(* CoDeSys 2.3.9.25 project: fuel_oil_v1.4.4.pro *)
(* Libraries: Util.lib 18.5.10 16:14:28, STANDARD.LIB 4.10.05 12:14:46, IECSFC.LIB 13.4.06 16:51:28, ANALYZATION.LIB 5.10.99 10:05:06 *)

(* PLC configuration (modules and I/O channels)
Fast discrete inputs [I_SIMPLE_INPUT] node 0, in %IB0 out %QB0 {Filtrationtime = 10; Visibility = No}
  AT %IX0.0 [BitInput] Discrete input 1
  AT %IX0.1 [BitInput] Discrete input 2
Discrete inputs - 16 [ID130] node 1, in %IB1 out %QB1 {Filtrationtime_GeneralINP = 1; Visibility = No; PinCount = 16}
  AT %IB1.0 [ByteInput] 8 discrete inputs
  AT %IB1.1 [ByteInput] 8 discrete inputs
Fast discrete outputs [OWEN_ID570] node 2, in %IB2 out %QB2 {SafeValueBool = FALSE; SafeValueBool = FALSE; SafeValueBool = FALSE; SafeValueBool = FALSE; Visibility = No}
  AT %QX2.0 [BitOutput] go_emul
  AT %QX2.1 [BitOutput] go_mixing
  AT %QX2.2 [BitOutput] go_diesel_bio
  AT %QX2.3 [BitOutput] go_water
AT %QB3.0 [ByteOutput] 8 discrete outputs
AT %QB3.1 [ByteOutput] 2 discrete outputs
Special input [ID103] node 4, in %IB4 out %QB4 {Filtrationtime = 1000; PinCount = 1; WatchDogPeriod = 400; PollPeriod = 3000; Visibility = No}
  AT %IX4.0 [BitInput] Special input
Special output [ID104] node 5, in %IB5 out %QB5 {Visibility = No; PinCount = 1}
  AT %QX5.0 [BitOutput] Special output
ModBus (Master) [MODBUS_MASTER_ID450] node 6, in %IB6 out %QB6 {Visibility = No}
  AT %QD6.0 [DWordOutput] Last address
  AT %QW6.1 [WordOutput] Last error
  RS-485-1 [COM1_USART] node 0, in %IB6.0 out %QB6.0 {CommunicationSpeed = 11520; Parity = NO PARITY CHECK; BitLength = 8 bits; StopLength = One stop bit; InterfaceType = RS485; FrameOriented = RTU; Timeout = 0; Visibility = No}
AT %QB6.1.0 [ComChannel] Command (0xff - Start)
AT %IW6.1.0.0 [WordInput]
AT %ID6.1.1.0 [FloatInput]
TCP [TCP_ID221] node 0, in %IB7.0.0 out %QB7.0.0 {RemotePort = 502; Visibility = No}
AT %QB7.1.0 [ByteOutput]
AT %QB7.2.0 [ByteOutput]
AT %QW7.3.0 [WordOutput] flow_out
AT %QW7.4.0 [WordOutput] weight_of_emul_LAN
AT %QW7.5.0 [WordOutput] weight_of_diesel_LAN
AT %QW7.6.0 [WordOutput] weight_of_biodiesel_LAN
AT %QW7.7.0 [WordOutput] set_number_of_liters_LAN
AT %QW7.8.0 [WordOutput] time_of_mixing_first
AT %QW7.9.0 [WordOutput] weight_left_LAN
AT %QW7.10.0 [WordOutput] empty
AT %QW7.11.0 [WordOutput] empty
AT %QW7.12.0 [WordOutput] avto_LAN
AT %QW7.13.0 [WordOutput] number_of_liters_LAN
AT %QW7.14.0 [WordOutput] time_of_mixing_second
AT %QW7.15.0 [WordOutput] pusk_LAN
AT %QW7.16.0 [WordOutput] stop_LAN
AT %QD7.17.0 [FloatOutput] wight_in_barrel_LAN
AT %QD7.18.0 [FloatOutput] wight_in_barrel_for_proc
AT %QD7.19.0 [FloatOutput] wight_for_sub_2
*)

(* POU PLC_PRG, LD *)
PROGRAM PLC_PRG
VAR
(*блок запуска/остоновки/паузы*)
	psp: psp;
	pusk AT %IX1.0.1: BOOL; (*сигнал на запуск цикла*)
	pusk_LAN AT %QW7.15.0: BOOL; (*сигнал на запуск цикла со SCADA*)
	avto AT %IX1.0.3: BOOL; (*перевод системы в автоматический режим*)
	stop AT %IX1.0.2: BOOL; (*сигнал на остановку цикла*)
	stop_LAN AT %QW7.16.0: BOOL; (*сигнал на остановку цикла со SCADA*)
	pusk_prog: BOOL; (*цикл запущен*)
	stop_prog AT %QX7.1.0.0: BOOL; (*цикл остановлен*)
	pause: BOOL; (*цикл поставлен на паузу*)
	wight_in_barrel AT %ID6.1.1.0: REAL; (*вес в баке, приходящий с весов*)
	work_lamp AT %QX3.0.3: BOOL; (*выходная лампа сигнализации работы*)
	wight_in_barrel_for_proc AT %QD7.18.0: REAL; (*количество кг смеси для цикла*)
	flow_reley AT %IX1.1.4: BOOL; (*срабатывание реле протока*)
	TZ2_LAN AT %QX7.1.0.3: BOOL;
	TZ3_LAN AT %QX7.1.0.4: BOOL;
	TZ4_LAN AT %QX7.1.0.5: BOOL;
	TZ5_LAN AT %QX7.1.0.6: BOOL;
	TZ6_LAN AT %QX7.1.0.7: BOOL;
	TZ7_LAN AT %QX7.2.0.0: BOOL;
	work_lamp_LAN AT %QX7.2.0.1: BOOL; (*лампа работы для Scada*)
	wight_in_barrel_LAN AT %QD7.17.0: REAL; (*значение текущего ввеса в баке для Scada*)
	for_setpoints: REAL; (*значения для рассчета аозможности перелива*)

(*блок предотвращения перелива жидкости из бака*)
	sum_of_setpoints: sum_of_setpoints;
	more_then_need AT %QX7.2.0.2: BOOL; (*сигнализации о том, что может произойти перелив*)

(*Блок для отправки значений работы насосов в Scada*)
	move_block: move_block;
	go_emul_LAN AT %QX7.2.0.3: BOOL;
	go_diesel_bio_LAN AT %QX7.2.0.4: BOOL;
	go_water_LAN AT %QX7.2.0.5: BOOL;
	go_mixing_LAN AT %QX7.2.0.6: BOOL;
	go_disper_LAN AT %QX7.2.0.7: BOOL;
	avto_LAN AT %QW7.12.0: BOOL;

(*блок запуска процесса наполнения бака эмульсией*)
	emul: emul;
	go_emul AT %QX2.0: BOOL; (*сигнал на запуск насоса эмульсии*)
	end_work_emul: BOOL; (*блок работы насоса эмульсии завершен*)
	flow_out: BOOL; (*реле протока не сработало*)
	flow_out_LAN AT %QW7.3.0: BOOL;

(*блок запуска насоса дизель/биодизель*)
	dies_bio: dies_bio;
	go_diesel_bio AT %QX2.2: BOOL; (*сигнал на запуск насоса дизель/биодизель*)
	stop_diesel: BOOL; (*сигнал о том что, наполнение дизеля в бак окончено*)
	end_work_dies_bio AT %QX7.1.0.1: BOOL; (*блок работы насоса дизель/биодизель завершен*)
	weight_next_step: REAL; (*количество жидкости для продолжения цикла*)
	both_null: BOOL;

(*блок запуска насоса воды*)
	water: water;
	count AT %IX0.0: BOOL; (*импульсы, приходящие со счетчика воды*)
	number_of_liters_LAN AT %QW7.13.0: WORD; (*количество воды, посчитанное счетчиком воды*)
	go_water AT %QX2.3: BOOL; (*сигнал на запуск насоса воды*)
	end_work_water: BOOL; (*блок работы насоса воды завершен*)
	go_valve AT %QX3.0.5: BOOL;

(*блок управлени насосом смешивания*)
	mixing: mixing;
	go_mixing AT %QX2.1: BOOL; (*сигнал на запуск насоса смешивания*)
	end_work_mixing: BOOL; (*блок работы насоса смешивания завершен*)
	end_work_first AT %QX7.1.0.2: BOOL; (*блок работы насоса завершил первое перемешивание*)

(*блок управления насосом диспергации*)
	disper: disper;
	go_disper AT %QX3.0.0: BOOL; (*сигнал на запуск насоса смешивания*)
	end_work_disper: BOOL; (*блок работы насоса диспергации завершен*)

	TZ2 AT %IX1.0.6: BOOL;
	TZ3 AT %IX1.0.7: BOOL;
	TZ4 AT %IX1.1.0: BOOL;
	TZ5 AT %IX1.1.1: BOOL;
	TZ6 AT %IX1.1.2: BOOL;
	TZ7 AT %IX1.1.3: BOOL;
	avar_TZ: BOOL; (*сработала одна из тепловых защит*)
	weight_of_diesel_for_mix: BOOL;

	for_calculate: CTU;
	calc_trig: R_TRIG;
	wight_for_sub_1: REAL;
	wight_for_sub_2 AT %QD7.19.0: REAL;
END_VAR

VAR RETAIN PERSISTENT
	weight_of_emul_LAN AT %QW7.4.0: WORD; (*количество эмульгатора для наполнения в бак, задается из SCADA*)
	weight_of_diesel_LAN AT %QW7.5.0: WORD; (*количество дизеля для наполнения в бак, задается из SCADA*)
	weight_of_biodiesel_LAN AT %QW7.6.0: WORD; (*количество биодизеля для наполнения в бак, задается из SCADA*)
	set_number_of_liters_LAN AT %QW7.7.0: WORD; (*количество воды для наполнения в бак, задается из SCADA*)
	time_of_mixing_first AT %QW7.8.0: WORD; (*время первого смешивания*)
	weight_left_LAN AT %QW7.9.0: WORD; (*колличество, которое должно остаться в баке после диспергации*)
	time_of_mixing_second AT %QW7.14.0: WORD; (*время второго смешивания*)
END_VAR
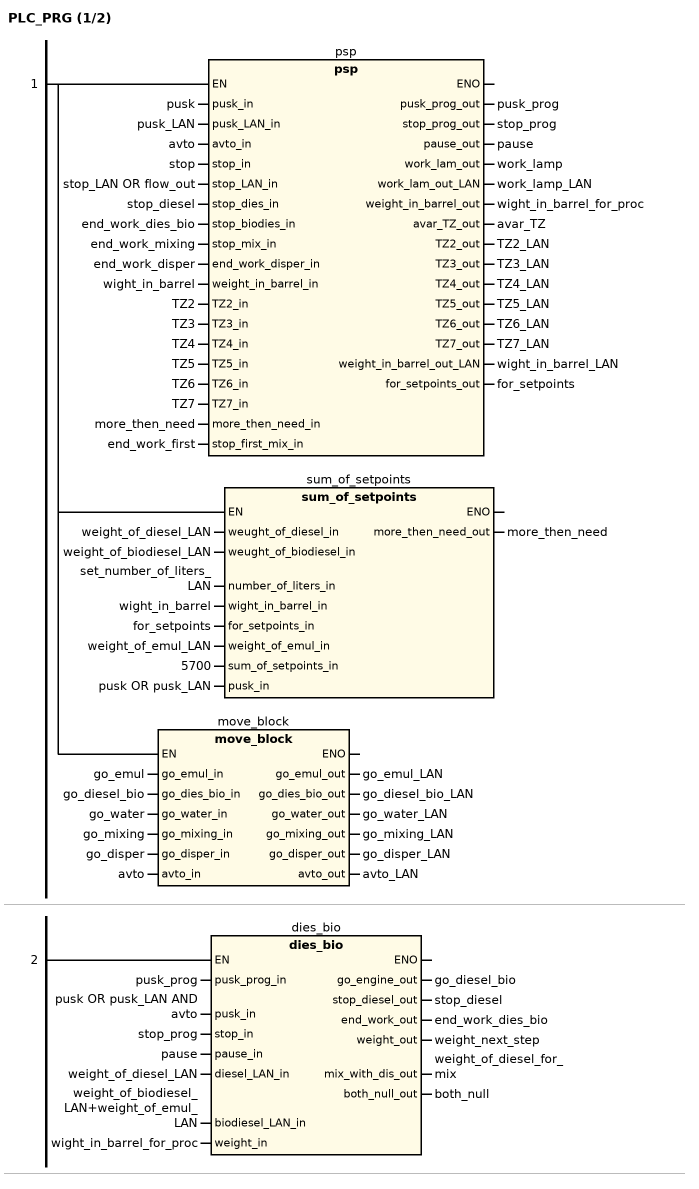
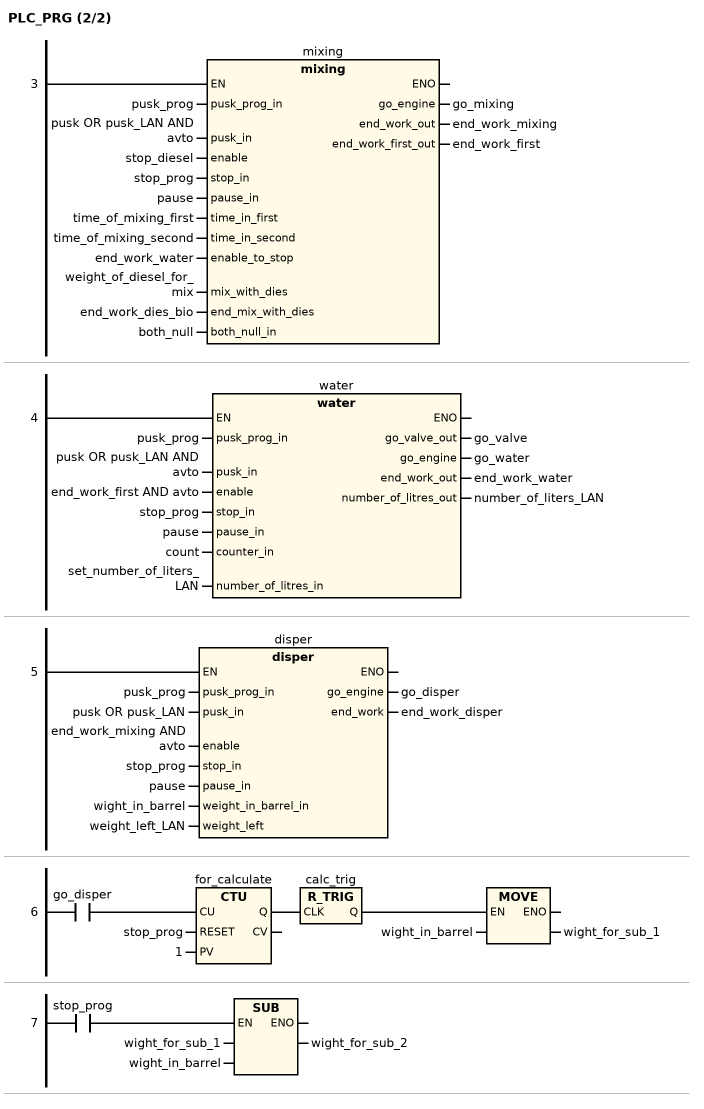
_LD_ (* Ladder Diagram *)
NETWORK 1
	*
		EN --- psp:psp(pusk_in: pusk, pusk_LAN_in: pusk_LAN, avto_in: avto, stop_in: stop, stop_LAN_in: stop_LAN OR flow_out, stop_dies_in: stop_diesel, stop_biodies_in: end_work_dies_bio, stop_mix_in: end_work_mixing, end_work_disper_in: end_work_disper, weight_in_barrel_in: wight_in_barrel, TZ2_in: TZ2, TZ3_in: TZ3, TZ4_in: TZ4, TZ5_in: TZ5, TZ6_in: TZ6, TZ7_in: TZ7, more_then_need_in: more_then_need, stop_first_mix_in: end_work_first, stop_prog_out => stop_prog, pause_out => pause, work_lam_out => work_lamp, work_lam_out_LAN => work_lamp_LAN, weight_in_barrel_out => wight_in_barrel_for_proc, avar_TZ_out => avar_TZ, TZ2_out => TZ2_LAN, TZ3_out => TZ3_LAN, TZ4_out => TZ4_LAN, TZ5_out => TZ5_LAN, TZ6_out => TZ6_LAN, TZ7_out => TZ7_LAN, weight_in_barrel_out_LAN => wight_in_barrel_LAN, for_setpoints_out => for_setpoints) => pusk_prog
		EN --- sum_of_setpoints:sum_of_setpoints(weught_of_diesel_in: weight_of_diesel_LAN, weught_of_biodiesel_in: weight_of_biodiesel_LAN, number_of_liters_in: set_number_of_liters_LAN, wight_in_barrel_in: wight_in_barrel, for_setpoints_in: for_setpoints, weight_of_emul_in: weight_of_emul_LAN, sum_of_setpoints_in: 5700, pusk_in: pusk OR pusk_LAN) => more_then_need
		EN --- move_block:move_block(go_emul_in: go_emul, go_dies_bio_in: go_diesel_bio, go_water_in: go_water, go_mixing_in: go_mixing, go_disper_in: go_disper, avto_in: avto, go_dies_bio_out => go_diesel_bio_LAN, go_water_out => go_water_LAN, go_mixing_out => go_mixing_LAN, go_disper_out => go_disper_LAN, avto_out => avto_LAN) => go_emul_LAN
NETWORK 2
	*
		EN --- dies_bio:dies_bio(pusk_prog_in: pusk_prog, pusk_in: pusk OR pusk_LAN AND avto, stop_in: stop_prog, pause_in: pause, diesel_LAN_in: weight_of_diesel_LAN, biodiesel_LAN_in: weight_of_biodiesel_LAN+weight_of_emul_LAN, weight_in: wight_in_barrel_for_proc, stop_diesel_out => stop_diesel, end_work_out => end_work_dies_bio, weight_out => weight_next_step, mix_with_dis_out => weight_of_diesel_for_mix, both_null_out => both_null) => go_diesel_bio
NETWORK 3
	*
		EN --- mixing:mixing(pusk_prog_in: pusk_prog, pusk_in: pusk OR pusk_LAN AND avto, enable: stop_diesel, stop_in: stop_prog, pause_in: pause, time_in_first: time_of_mixing_first, time_in_second: time_of_mixing_second, enable_to_stop: end_work_water, mix_with_dies: weight_of_diesel_for_mix, end_mix_with_dies: end_work_dies_bio, both_null_in: both_null, end_work_out => end_work_mixing, end_work_first_out => end_work_first) => go_mixing
NETWORK 4
	*
		EN --- water:water(pusk_prog_in: pusk_prog, pusk_in: pusk OR pusk_LAN AND avto, enable: end_work_first AND avto, stop_in: stop_prog, pause_in: pause, counter_in: count, number_of_litres_in: set_number_of_liters_LAN, go_engine => go_water, end_work_out => end_work_water, number_of_litres_out => number_of_liters_LAN) => go_valve
NETWORK 5
	*
		EN --- disper:disper(pusk_prog_in: pusk_prog, pusk_in: pusk OR pusk_LAN, enable: end_work_mixing AND avto, stop_in: stop_prog, pause_in: pause, weight_in_barrel_in: wight_in_barrel, weight_left: weight_left_LAN, end_work => end_work_disper) => go_disper
NETWORK 6
	[go_disper] - for_calculate:CTU(CU: *, RESET: stop_prog, PV: 1) - calc_trig:R_TRIG(CLK: *)
		EN --- MOVE(wight_in_barrel) => wight_for_sub_1
NETWORK 7
	[stop_prog]
		EN --- SUB(wight_for_sub_1, wight_in_barrel) => wight_for_sub_2
_END_LD_
(* the same logic as Structured Text *)
(* Network 1 *)
psp(pusk_in := pusk, pusk_LAN_in := pusk_LAN, avto_in := avto, stop_in := stop, stop_LAN_in := stop_LAN OR flow_out, stop_dies_in := stop_diesel, stop_biodies_in := end_work_dies_bio, stop_mix_in := end_work_mixing, end_work_disper_in := end_work_disper, weight_in_barrel_in := wight_in_barrel, TZ2_in := TZ2, TZ3_in := TZ3, TZ4_in := TZ4, TZ5_in := TZ5, TZ6_in := TZ6, TZ7_in := TZ7, more_then_need_in := more_then_need, stop_first_mix_in := end_work_first);
stop_prog := psp.stop_prog_out;
pause := psp.pause_out;
work_lamp := psp.work_lam_out;
work_lamp_LAN := psp.work_lam_out_LAN;
wight_in_barrel_for_proc := psp.weight_in_barrel_out;
avar_TZ := psp.avar_TZ_out;
TZ2_LAN := psp.TZ2_out;
TZ3_LAN := psp.TZ3_out;
TZ4_LAN := psp.TZ4_out;
TZ5_LAN := psp.TZ5_out;
TZ6_LAN := psp.TZ6_out;
TZ7_LAN := psp.TZ7_out;
wight_in_barrel_LAN := psp.weight_in_barrel_out_LAN;
for_setpoints := psp.for_setpoints_out;
pusk_prog := psp.pusk_prog_out;
sum_of_setpoints(weught_of_diesel_in := weight_of_diesel_LAN, weught_of_biodiesel_in := weight_of_biodiesel_LAN, number_of_liters_in := set_number_of_liters_LAN, wight_in_barrel_in := wight_in_barrel, for_setpoints_in := for_setpoints, weight_of_emul_in := weight_of_emul_LAN, sum_of_setpoints_in := 5700, pusk_in := pusk OR pusk_LAN);
more_then_need := sum_of_setpoints.more_then_need_out;
move_block(go_emul_in := go_emul, go_dies_bio_in := go_diesel_bio, go_water_in := go_water, go_mixing_in := go_mixing, go_disper_in := go_disper, avto_in := avto);
go_diesel_bio_LAN := move_block.go_dies_bio_out;
go_water_LAN := move_block.go_water_out;
go_mixing_LAN := move_block.go_mixing_out;
go_disper_LAN := move_block.go_disper_out;
avto_LAN := move_block.avto_out;
go_emul_LAN := move_block.go_emul_out;
(* Network 2 *)
dies_bio(pusk_prog_in := pusk_prog, pusk_in := pusk OR pusk_LAN AND avto, stop_in := stop_prog, pause_in := pause, diesel_LAN_in := weight_of_diesel_LAN, biodiesel_LAN_in := weight_of_biodiesel_LAN+weight_of_emul_LAN, weight_in := wight_in_barrel_for_proc);
stop_diesel := dies_bio.stop_diesel_out;
end_work_dies_bio := dies_bio.end_work_out;
weight_next_step := dies_bio.weight_out;
weight_of_diesel_for_mix := dies_bio.mix_with_dis_out;
both_null := dies_bio.both_null_out;
go_diesel_bio := dies_bio.go_engine_out;
(* Network 3 *)
mixing(pusk_prog_in := pusk_prog, pusk_in := pusk OR pusk_LAN AND avto, enable := stop_diesel, stop_in := stop_prog, pause_in := pause, time_in_first := time_of_mixing_first, time_in_second := time_of_mixing_second, enable_to_stop := end_work_water, mix_with_dies := weight_of_diesel_for_mix, end_mix_with_dies := end_work_dies_bio, both_null_in := both_null);
end_work_mixing := mixing.end_work_out;
end_work_first := mixing.end_work_first_out;
go_mixing := mixing.go_engine;
(* Network 4 *)
water(pusk_prog_in := pusk_prog, pusk_in := pusk OR pusk_LAN AND avto, enable := end_work_first AND avto, stop_in := stop_prog, pause_in := pause, counter_in := count, number_of_litres_in := set_number_of_liters_LAN);
go_water := water.go_engine;
end_work_water := water.end_work_out;
number_of_liters_LAN := water.number_of_litres_out;
go_valve := water.go_valve_out;
(* Network 5 *)
disper(pusk_prog_in := pusk_prog, pusk_in := pusk OR pusk_LAN, enable := end_work_mixing AND avto, stop_in := stop_prog, pause_in := pause, weight_in_barrel_in := wight_in_barrel, weight_left := weight_left_LAN);
end_work_disper := disper.end_work;
go_disper := disper.go_engine;
(* Network 6 *)
for_calculate(CU := go_disper, RESET := stop_prog, PV := 1);
calc_trig(CLK := for_calculate.Q);
IF calc_trig.Q THEN
	wight_for_sub_1 := wight_in_barrel;
END_IF;
(* Network 7 *)
IF stop_prog THEN
	wight_for_sub_2 := wight_for_sub_1 - wight_in_barrel;
END_IF;
END_PROGRAM

(* POU psp, LD *)
FUNCTION_BLOCK psp (*блок пуска-остановки программы цикла, а так же установки цикла на пауза*)
VAR_INPUT
	pusk_in: BOOL;
	pusk_LAN_in: BOOL;
	avto_in: BOOL;
	stop_in: BOOL;
	stop_LAN_in: BOOL;
	stop_dies_in: BOOL;
	stop_biodies_in: BOOL;
	stop_mix_in: BOOL;
	end_work_disper_in: BOOL;
	weight_in_barrel_in: REAL;
	TZ2_in: BOOL;
	TZ3_in: BOOL;
	TZ4_in: BOOL;
	TZ5_in: BOOL;
	TZ6_in: BOOL;
	TZ7_in: BOOL;
	more_then_need_in: BOOL;
	stop_first_mix_in: BOOL;
END_VAR
VAR_OUTPUT
	pusk_prog_out: BOOL;
	stop_prog_out: BOOL;
	pause_out: BOOL;
	work_lam_out: BOOL;
	work_lam_out_LAN: BOOL;
	weight_in_barrel_out: REAL;
	avar_TZ_out: BOOL;
	TZ2_out: BOOL;
	TZ3_out: BOOL;
	TZ4_out: BOOL;
	TZ5_out: BOOL;
	TZ6_out: BOOL;
	TZ7_out: BOOL;
	weight_in_barrel_out_LAN: REAL;
	for_setpoints_out: REAL;
END_VAR
VAR
	rs1: RS;
	ctu1: CTU;
	pause_ins: BOOL;
	ctu2: CTU;
	blink1: BLINK;
	pause_blink: BOOL;
	rtr1: R_TRIG;
	stop_prog_ins: BOOL;
	tp1: TP;
	rtr2: R_TRIG;
	rtr3: R_TRIG;
	ftr1: F_TRIG;
	more_then_need_ins: BOOL;
	tp2: TP;
	weight_in_barrel_ins: REAL;
	rtr4: R_TRIG;
	rtr5: R_TRIG;
END_VAR
VAR (* helpers for the ST form of the networks *)
	_p1 : BOOL;
	_p2 : BOOL;
END_VAR
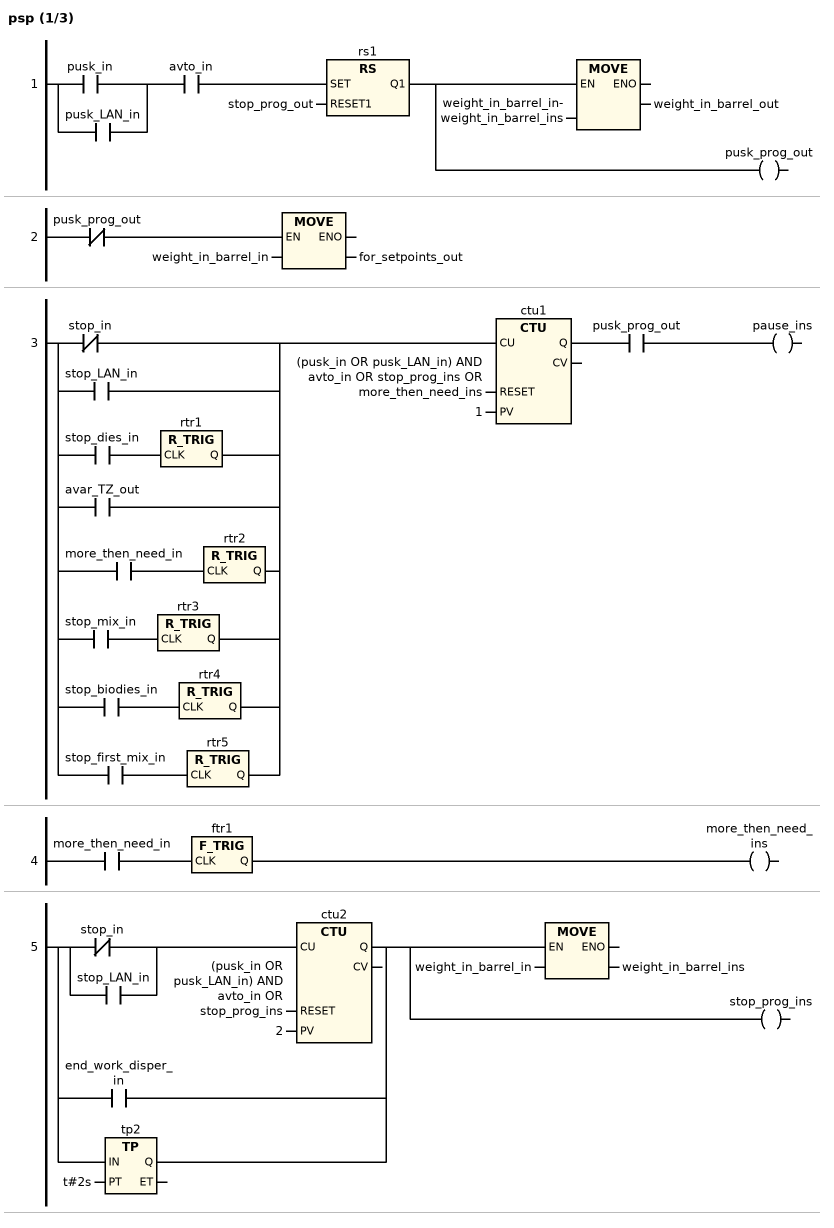
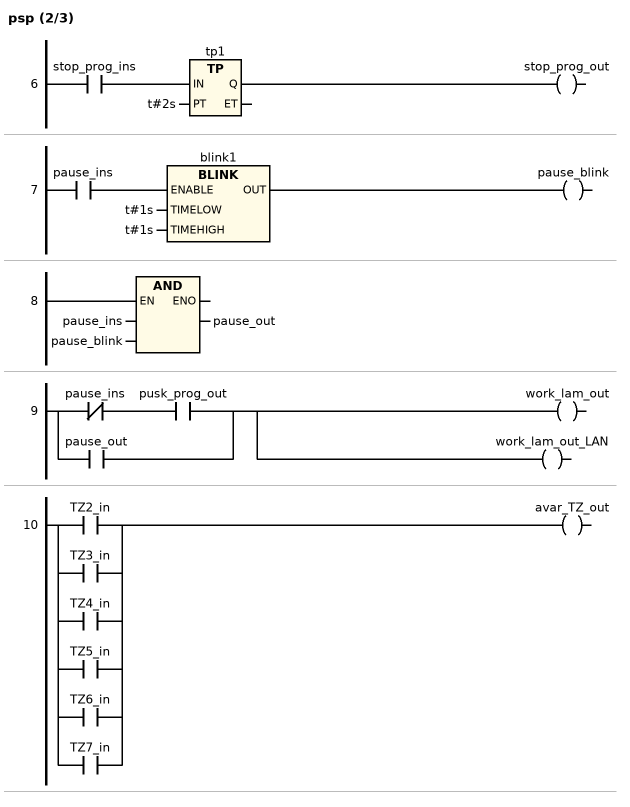
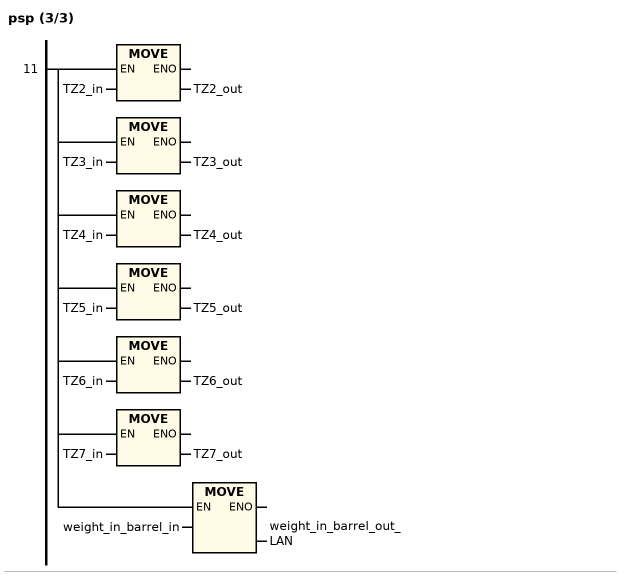
_LD_ (* Ladder Diagram *)
NETWORK 1
	{ [pusk_in] | [pusk_LAN_in] } - [avto_in] - rs1:RS(SET: *, RESET1: stop_prog_out) --- (pusk_prog_out)
		EN --- MOVE(weight_in_barrel_in-weight_in_barrel_ins) => weight_in_barrel_out
NETWORK 2
	[/pusk_prog_out]
		EN --- MOVE(weight_in_barrel_in) => for_setpoints_out
NETWORK 3
	{ [/stop_in] | [stop_LAN_in] | [stop_dies_in] - rtr1:R_TRIG(CLK: *) | [avar_TZ_out] | [more_then_need_in] - rtr2:R_TRIG(CLK: *) | [stop_mix_in] - rtr3:R_TRIG(CLK: *) | [stop_biodies_in] - rtr4:R_TRIG(CLK: *) | [stop_first_mix_in] - rtr5:R_TRIG(CLK: *) } - ctu1:CTU(CU: *, RESET: (pusk_in OR pusk_LAN_in) AND avto_in OR stop_prog_ins OR more_then_need_ins, PV: 1) - [pusk_prog_out] --- (pause_ins)
NETWORK 4
	[more_then_need_in] - ftr1:F_TRIG(CLK: *) --- (more_then_need_ins)
NETWORK 5
	{ { [/stop_in] | [stop_LAN_in] } - ctu2:CTU(CU: *, RESET: (pusk_in OR pusk_LAN_in) AND avto_in OR stop_prog_ins, PV: 2) | [end_work_disper_in] | tp2:TP(IN: *, PT: t#2s) } --- (stop_prog_ins)
		EN --- MOVE(weight_in_barrel_in) => weight_in_barrel_ins
NETWORK 6
	[stop_prog_ins] - tp1:TP(IN: *, PT: t#2s) --- (stop_prog_out)
NETWORK 7
	[pause_ins] - blink1:BLINK(ENABLE: *, TIMELOW: t#1s, TIMEHIGH: t#1s) --- (pause_blink)
NETWORK 8
	*
		EN --- AND(pause_ins, pause_blink) => pause_out
NETWORK 9
	{ [/pause_ins] - [pusk_prog_out] | [pause_out] } --- (work_lam_out) (work_lam_out_LAN)
NETWORK 10
	{ [TZ2_in] | [TZ3_in] | [TZ4_in] | [TZ5_in] | [TZ6_in] | [TZ7_in] } --- (avar_TZ_out)
NETWORK 11
	*
		EN --- MOVE(TZ2_in) => TZ2_out
		EN --- MOVE(TZ3_in) => TZ3_out
		EN --- MOVE(TZ4_in) => TZ4_out
		EN --- MOVE(TZ5_in) => TZ5_out
		EN --- MOVE(TZ6_in) => TZ6_out
		EN --- MOVE(TZ7_in) => TZ7_out
		EN --- MOVE(weight_in_barrel_in) => weight_in_barrel_out_LAN
_END_LD_
(* the same logic as Structured Text *)
(* Network 1 *)
rs1(SET := (pusk_in OR pusk_LAN_in) AND avto_in, RESET1 := stop_prog_out);
_p1 := rs1.Q1;
IF _p1 THEN
	weight_in_barrel_out := weight_in_barrel_in-weight_in_barrel_ins;
END_IF;
pusk_prog_out := _p1;
(* Network 2 *)
IF NOT pusk_prog_out THEN
	for_setpoints_out := weight_in_barrel_in;
END_IF;
(* Network 3 *)
rtr1(CLK := stop_dies_in);
rtr2(CLK := more_then_need_in);
rtr3(CLK := stop_mix_in);
rtr4(CLK := stop_biodies_in);
rtr5(CLK := stop_first_mix_in);
ctu1(CU := NOT stop_in OR stop_LAN_in OR rtr1.Q OR avar_TZ_out OR rtr2.Q OR rtr3.Q OR rtr4.Q OR rtr5.Q, RESET := (pusk_in OR pusk_LAN_in) AND avto_in OR stop_prog_ins OR more_then_need_ins, PV := 1);
pause_ins := ctu1.Q AND pusk_prog_out;
(* Network 4 *)
ftr1(CLK := more_then_need_in);
more_then_need_ins := ftr1.Q;
(* Network 5 *)
ctu2(CU := NOT stop_in OR stop_LAN_in, RESET := (pusk_in OR pusk_LAN_in) AND avto_in OR stop_prog_ins, PV := 2);
tp2(IN := TRUE, PT := t#2s);
_p2 := ctu2.Q OR end_work_disper_in OR tp2.Q;
IF _p2 THEN
	weight_in_barrel_ins := weight_in_barrel_in;
END_IF;
stop_prog_ins := _p2;
(* Network 6 *)
tp1(IN := stop_prog_ins, PT := t#2s);
stop_prog_out := tp1.Q;
(* Network 7 *)
blink1(ENABLE := pause_ins, TIMELOW := t#1s, TIMEHIGH := t#1s);
pause_blink := blink1.OUT;
(* Network 8 *)
pause_out := pause_ins AND pause_blink;
(* Network 9 *)
work_lam_out := NOT pause_ins AND pusk_prog_out OR pause_out;
work_lam_out_LAN := work_lam_out;
(* Network 10 *)
avar_TZ_out := TZ2_in OR TZ3_in OR TZ4_in OR TZ5_in OR TZ6_in OR TZ7_in;
(* Network 11 *)
TZ2_out := TZ2_in;
TZ3_out := TZ3_in;
TZ4_out := TZ4_in;
TZ5_out := TZ5_in;
TZ6_out := TZ6_in;
TZ7_out := TZ7_in;
weight_in_barrel_out_LAN := weight_in_barrel_in;
END_FUNCTION_BLOCK

(* POU sum_of_setpoints, FBD *)
FUNCTION_BLOCK sum_of_setpoints (*Блок рассчета вероятности перелива*)
VAR_INPUT
	weught_of_diesel_in: WORD;
	weught_of_biodiesel_in: WORD;
	number_of_liters_in: WORD;
	wight_in_barrel_in: REAL;
	for_setpoints_in: REAL;
	weight_of_emul_in: WORD;
	sum_of_setpoints_in: WORD;
	pusk_in: BOOL;
END_VAR
VAR_OUTPUT
	more_then_need_out: BOOL;
END_VAR
VAR
	sum_of_setpoints_ins: REAL;
	koef: REAL := 0.855;
	weught_of_diesel_real: REAL;
	weught_of_biodiesel_real: REAL;
END_VAR
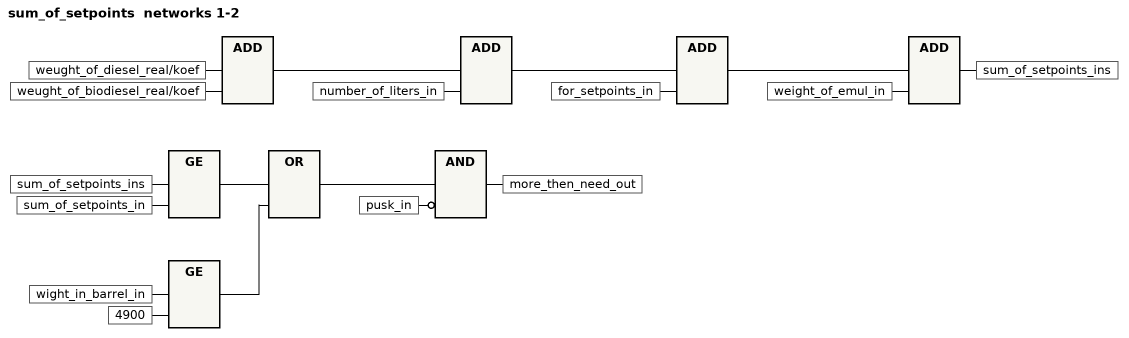
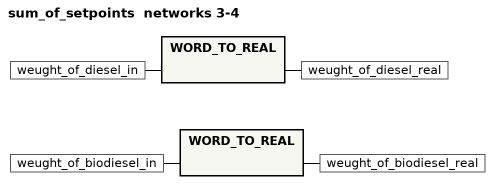
_FBD_ (* Function Block Diagram *)
NETWORK 1
	ADD(ADD(ADD(ADD(weught_of_diesel_real/koef, weught_of_biodiesel_real/koef), number_of_liters_in), for_setpoints_in), weight_of_emul_in) => sum_of_setpoints_ins
NETWORK 2
	AND(OR(GE(sum_of_setpoints_ins, sum_of_setpoints_in), GE(wight_in_barrel_in, 4900)), NOT pusk_in) => more_then_need_out
NETWORK 3
	WORD_TO_REAL(weught_of_diesel_in) => weught_of_diesel_real
NETWORK 4
	WORD_TO_REAL(weught_of_biodiesel_in) => weught_of_biodiesel_real
_END_FBD_
(* the same logic as Structured Text *)
(* Network 1 *)
sum_of_setpoints_ins := ((((weught_of_diesel_real/koef) + (weught_of_biodiesel_real/koef)) + number_of_liters_in) + for_setpoints_in) + weight_of_emul_in;
(* Network 2 *)
more_then_need_out := ((sum_of_setpoints_ins >= sum_of_setpoints_in) OR (wight_in_barrel_in >= 4900)) AND NOT pusk_in;
(* Network 3 *)
weught_of_diesel_real := WORD_TO_REAL(weught_of_diesel_in);
(* Network 4 *)
weught_of_biodiesel_real := WORD_TO_REAL(weught_of_biodiesel_in);
END_FUNCTION_BLOCK

(* POU move_block, LD *)
FUNCTION_BLOCK move_block (*блок-клемник для отправки значений в Scada*)
VAR_INPUT
	go_emul_in: BOOL;
	go_dies_bio_in: BOOL;
	go_water_in: BOOL;
	go_mixing_in: BOOL;
	go_disper_in: BOOL;
	avto_in: BOOL;
END_VAR
VAR_OUTPUT
	go_emul_out: BOOL;
	go_dies_bio_out: BOOL;
	go_water_out: BOOL;
	go_mixing_out: BOOL;
	go_disper_out: BOOL;
	avto_out: BOOL;
END_VAR
VAR
END_VAR
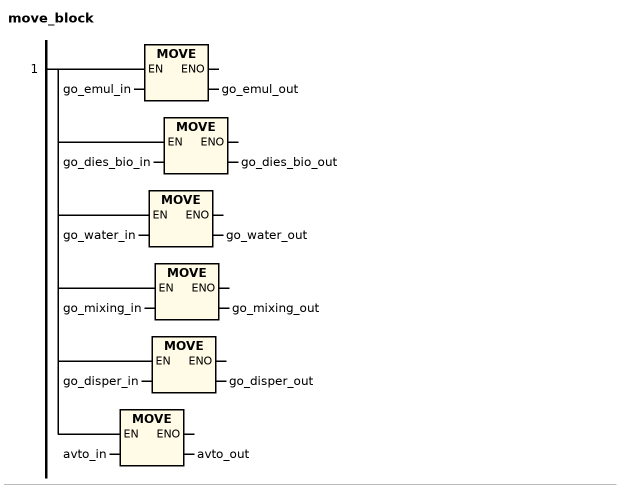
_LD_ (* Ladder Diagram *)
NETWORK 1
	*
		EN --- MOVE(go_emul_in) => go_emul_out
		EN --- MOVE(go_dies_bio_in) => go_dies_bio_out
		EN --- MOVE(go_water_in) => go_water_out
		EN --- MOVE(go_mixing_in) => go_mixing_out
		EN --- MOVE(go_disper_in) => go_disper_out
		EN --- MOVE(avto_in) => avto_out
_END_LD_
(* the same logic as Structured Text *)
(* Network 1 *)
go_emul_out := go_emul_in;
go_dies_bio_out := go_dies_bio_in;
go_water_out := go_water_in;
go_mixing_out := go_mixing_in;
go_disper_out := go_disper_in;
avto_out := avto_in;
END_FUNCTION_BLOCK

(* POU emul, LD *)
FUNCTION_BLOCK emul (*Блок работы насоса эмульгатора(дозировки)*)
VAR_INPUT
	pusk_prog_in:BOOL;
	pusk_in: BOOL;
	enable: BOOL;
	stop_in: BOOL;
	pause_in: BOOL;
	weight_in: REAL;
	flow_reley_in: BOOL;
	emul_LAN_in: WORD;
	weight_in_barel_in: REAL;
END_VAR
VAR_OUTPUT
	go_engine: BOOL;
	end_work_out: BOOL;
	flow_reley_out: BOOL;
	flow_reley_out_LAN: BOOL;
END_VAR
VAR
	rs1: RS;
	ton1: TON;
	rs2: RS;
	rtr1: R_TRIG;
	rs3: RS;
	stop_emul: BOOL;
	rtr2: R_TRIG;
	rs4: RS;
	rtr3: R_TRIG;
	ton2: TON;
END_VAR
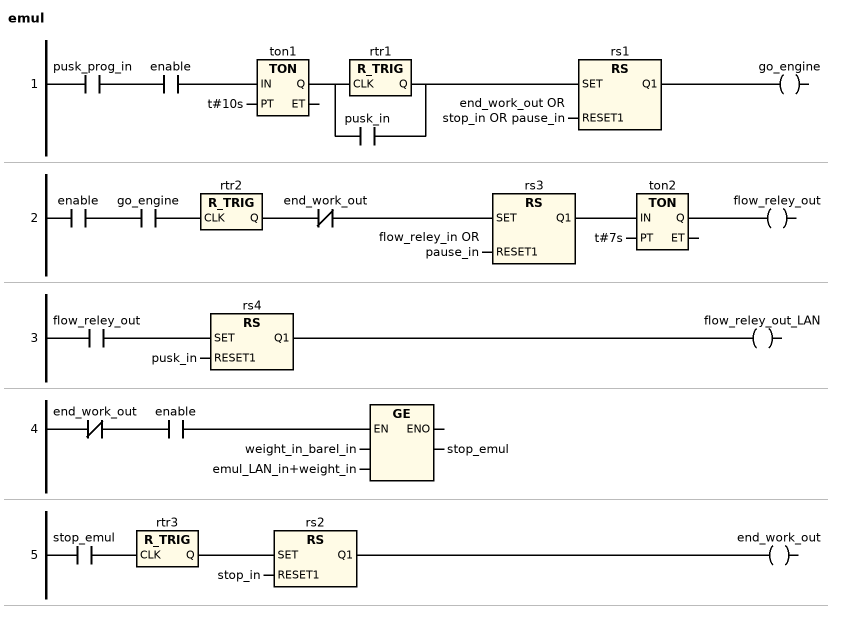
_LD_ (* Ladder Diagram *)
NETWORK 1
	[pusk_prog_in] - [enable] - ton1:TON(IN: *, PT: t#10s) - { rtr1:R_TRIG(CLK: *) | [pusk_in] } - rs1:RS(SET: *, RESET1: end_work_out OR stop_in OR pause_in) --- (go_engine)
NETWORK 2
	[enable] - [go_engine] - rtr2:R_TRIG(CLK: *) - [/end_work_out] - rs3:RS(SET: *, RESET1: flow_reley_in OR pause_in) - ton2:TON(IN: *, PT: t#7s) --- (flow_reley_out)
NETWORK 3
	[flow_reley_out] - rs4:RS(SET: *, RESET1: pusk_in) --- (flow_reley_out_LAN)
NETWORK 4
	[/end_work_out] - [enable]
		EN --- GE(weight_in_barel_in, emul_LAN_in+weight_in) => stop_emul
NETWORK 5
	[stop_emul] - rtr3:R_TRIG(CLK: *) - rs2:RS(SET: *, RESET1: stop_in) --- (end_work_out)
_END_LD_
(* the same logic as Structured Text *)
(* Network 1 *)
ton1(IN := pusk_prog_in AND enable, PT := t#10s);
rtr1(CLK := ton1.Q);
rs1(SET := rtr1.Q OR ton1.Q AND pusk_in, RESET1 := end_work_out OR stop_in OR pause_in);
go_engine := rs1.Q1;
(* Network 2 *)
rtr2(CLK := enable AND go_engine);
rs3(SET := rtr2.Q AND NOT end_work_out, RESET1 := flow_reley_in OR pause_in);
ton2(IN := rs3.Q1, PT := t#7s);
flow_reley_out := ton2.Q;
(* Network 3 *)
rs4(SET := flow_reley_out, RESET1 := pusk_in);
flow_reley_out_LAN := rs4.Q1;
(* Network 4 *)
IF NOT end_work_out AND enable THEN
	stop_emul := weight_in_barel_in >= (emul_LAN_in+weight_in);
END_IF;
(* Network 5 *)
rtr3(CLK := stop_emul);
rs2(SET := rtr3.Q, RESET1 := stop_in);
end_work_out := rs2.Q1;
END_FUNCTION_BLOCK

(* POU dies_bio, LD *)
FUNCTION_BLOCK dies_bio (*Блок работы насоса дизель-биодизель*)
VAR_INPUT
	pusk_prog_in: BOOL;
	pusk_in: BOOL;
	stop_in: BOOL;
	pause_in: BOOL;
	diesel_LAN_in: WORD;
	biodiesel_LAN_in: WORD;
	weight_in: REAL;
END_VAR
VAR_OUTPUT
	go_engine_out: BOOL;
	stop_diesel_out: BOOL;
	end_work_out: BOOL;
	weight_out: REAL;
	mix_with_dis_out: BOOL;
	both_null_out: BOOL;
END_VAR
VAR
	rs1: RS;
	rtr1: R_TRIG;
	rtr2: R_TRIG;
	stop_biodiesel: BOOL;
	wieght_of_diesel: REAL;
	rs2: RS;
	rtr3: R_TRIG;
	tof1: TOF;

	diesel_LAN_null: BOOL;
	biodiesel_LAN_null: BOOL;

	r_trig_one_not_null: R_TRIG;
	one_not_null_q: BOOL;
	rtr10: R_TRIG;
END_VAR
VAR (* helpers for the ST form of the networks *)
	_p1 : BOOL;
END_VAR
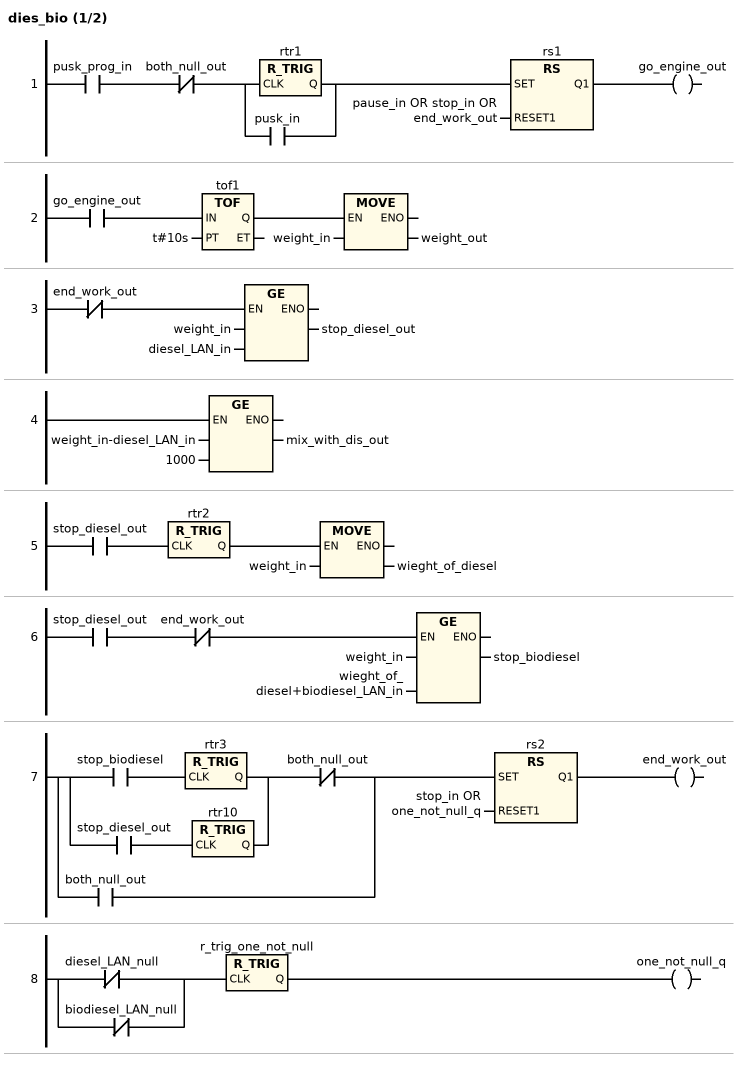
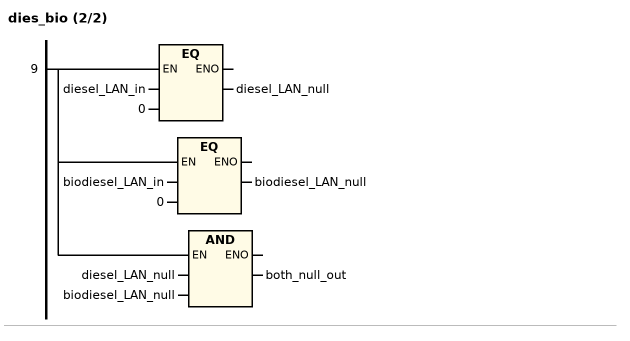
_LD_ (* Ladder Diagram *)
NETWORK 1
	[pusk_prog_in] - [/both_null_out] - { rtr1:R_TRIG(CLK: *) | [pusk_in] } - rs1:RS(SET: *, RESET1: pause_in OR stop_in OR end_work_out) --- (go_engine_out)
NETWORK 2
	[go_engine_out] - tof1:TOF(IN: *, PT: t#10s)
		EN --- MOVE(weight_in) => weight_out
NETWORK 3
	[/end_work_out]
		EN --- GE(weight_in, diesel_LAN_in) => stop_diesel_out
NETWORK 4
	*
		EN --- GE(weight_in-diesel_LAN_in, 1000) => mix_with_dis_out
NETWORK 5
	[stop_diesel_out] - rtr2:R_TRIG(CLK: *)
		EN --- MOVE(weight_in) => wieght_of_diesel
NETWORK 6
	[stop_diesel_out] - [/end_work_out]
		EN --- GE(weight_in, wieght_of_diesel+biodiesel_LAN_in) => stop_biodiesel
NETWORK 7
	{ { [stop_biodiesel] - rtr3:R_TRIG(CLK: *) | [stop_diesel_out] - rtr10:R_TRIG(CLK: *) } - [/both_null_out] | [both_null_out] } - rs2:RS(SET: *, RESET1: stop_in OR one_not_null_q) --- (end_work_out)
NETWORK 8
	{ [/diesel_LAN_null] | [/biodiesel_LAN_null] } - r_trig_one_not_null:R_TRIG(CLK: *) --- (one_not_null_q)
NETWORK 9
	*
		EN --- EQ(diesel_LAN_in, 0) => diesel_LAN_null
		EN --- EQ(biodiesel_LAN_in, 0) => biodiesel_LAN_null
		EN --- AND(diesel_LAN_null, biodiesel_LAN_null) => both_null_out
_END_LD_
(* the same logic as Structured Text *)
(* Network 1 *)
_p1 := pusk_prog_in AND NOT both_null_out;
rtr1(CLK := _p1);
rs1(SET := rtr1.Q OR _p1 AND pusk_in, RESET1 := pause_in OR stop_in OR end_work_out);
go_engine_out := rs1.Q1;
(* Network 2 *)
tof1(IN := go_engine_out, PT := t#10s);
IF tof1.Q THEN
	weight_out := weight_in;
END_IF;
(* Network 3 *)
IF NOT end_work_out THEN
	stop_diesel_out := weight_in >= diesel_LAN_in;
END_IF;
(* Network 4 *)
mix_with_dis_out := (weight_in-diesel_LAN_in) >= 1000;
(* Network 5 *)
rtr2(CLK := stop_diesel_out);
IF rtr2.Q THEN
	wieght_of_diesel := weight_in;
END_IF;
(* Network 6 *)
IF stop_diesel_out AND NOT end_work_out THEN
	stop_biodiesel := weight_in >= (wieght_of_diesel+biodiesel_LAN_in);
END_IF;
(* Network 7 *)
rtr3(CLK := stop_biodiesel);
rtr10(CLK := stop_diesel_out);
rs2(SET := (rtr3.Q OR rtr10.Q) AND NOT both_null_out OR both_null_out, RESET1 := stop_in OR one_not_null_q);
end_work_out := rs2.Q1;
(* Network 8 *)
r_trig_one_not_null(CLK := NOT diesel_LAN_null OR NOT biodiesel_LAN_null);
one_not_null_q := r_trig_one_not_null.Q;
(* Network 9 *)
diesel_LAN_null := diesel_LAN_in = 0;
biodiesel_LAN_null := biodiesel_LAN_in = 0;
both_null_out := diesel_LAN_null AND biodiesel_LAN_null;
END_FUNCTION_BLOCK

(* POU water, LD *)
FUNCTION_BLOCK water (*Блок работы насоса воды*)
VAR_INPUT
	pusk_prog_in: BOOL;
	pusk_in: BOOL;
	enable: BOOL;
	stop_in: BOOL;
	pause_in: BOOL;
	counter_in: BOOL;
	number_of_litres_in: WORD;
END_VAR
VAR_OUTPUT
	go_valve_out: BOOL;
	go_engine: BOOL;
	end_work_out: BOOL;
	number_of_litres_out: WORD;
END_VAR
VAR
	rtr1: R_TRIG;
	rs1: RS;
	ctu1: CTU;
	litres_full: BOOL;
	rs2: RS;
	rtr3: R_TRIG;
	ton1: TON;

	liter_null: BOOL;
END_VAR
VAR (* helpers for the ST form of the networks *)
	_p1 : BOOL;
END_VAR
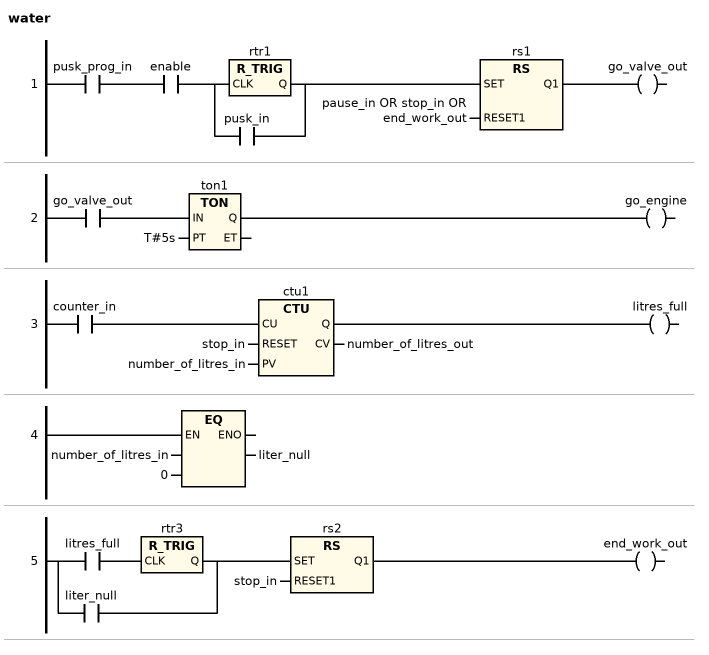
_LD_ (* Ladder Diagram *)
NETWORK 1
	[pusk_prog_in] - [enable] - { rtr1:R_TRIG(CLK: *) | [pusk_in] } - rs1:RS(SET: *, RESET1: pause_in OR stop_in OR end_work_out) --- (go_valve_out)
NETWORK 2
	[go_valve_out] - ton1:TON(IN: *, PT: T#5s) --- (go_engine)
NETWORK 3
	[counter_in] - ctu1:CTU(CU: *, RESET: stop_in, PV: number_of_litres_in, CV => number_of_litres_out) --- (litres_full)
NETWORK 4
	*
		EN --- EQ(number_of_litres_in, 0) => liter_null
NETWORK 5
	{ [litres_full] - rtr3:R_TRIG(CLK: *) | [liter_null] } - rs2:RS(SET: *, RESET1: stop_in) --- (end_work_out)
_END_LD_
(* the same logic as Structured Text *)
(* Network 1 *)
_p1 := pusk_prog_in AND enable;
rtr1(CLK := _p1);
rs1(SET := rtr1.Q OR _p1 AND pusk_in, RESET1 := pause_in OR stop_in OR end_work_out);
go_valve_out := rs1.Q1;
(* Network 2 *)
ton1(IN := go_valve_out, PT := T#5s);
go_engine := ton1.Q;
(* Network 3 *)
ctu1(CU := counter_in, RESET := stop_in, PV := number_of_litres_in);
number_of_litres_out := ctu1.CV;
litres_full := ctu1.Q;
(* Network 4 *)
liter_null := number_of_litres_in = 0;
(* Network 5 *)
rtr3(CLK := litres_full);
rs2(SET := rtr3.Q OR liter_null, RESET1 := stop_in);
end_work_out := rs2.Q1;
END_FUNCTION_BLOCK

(* POU mixing, LD *)
FUNCTION_BLOCK mixing (*Блок работы насоса смешивания*)
VAR_INPUT
	pusk_prog_in: BOOL;
	pusk_in: BOOL;
	enable: BOOL;
	stop_in: BOOL;
	pause_in: BOOL;
	time_in_first: WORD;
	time_in_second: WORD;
	enable_to_stop: BOOL;
	mix_with_dies: BOOL;
	end_mix_with_dies: BOOL;
	both_null_in: BOOL;
END_VAR
VAR_OUTPUT
	go_engine: BOOL;
	end_work_out: BOOL;
	end_work_first_out: BOOL;
END_VAR
VAR
	rs1: RS;
	ton1: TON;
	timer_off_first: BOOL;
	rs2: RS;
	rtr1: R_TRIG;
	ftr1: F_TRIG;
	run_time1: TIME;
	div_time1: TIME;
	run_time2: TIME;
	div_time2: TIME;
	sum_time1: TIME;
	sum_time2: TIME;
	time_ins1: DWORD;
	work_time1: TIME;
	time_ins2: DWORD;
	work_time2: TIME;
	ton2: TON;
	timer_off_second: BOOL;
	rs3: RS;
	rtr2: R_TRIG;
	end_mix_with_dies_ins: BOOL;

	end_mix_without_dies: BOOL;
	run1_more: BOOL;
	sum1_more: BOOL;
END_VAR
VAR (* helpers for the ST form of the networks *)
	_p1 : BOOL;
	_p2 : BOOL;
	_p3 : BOOL;
END_VAR
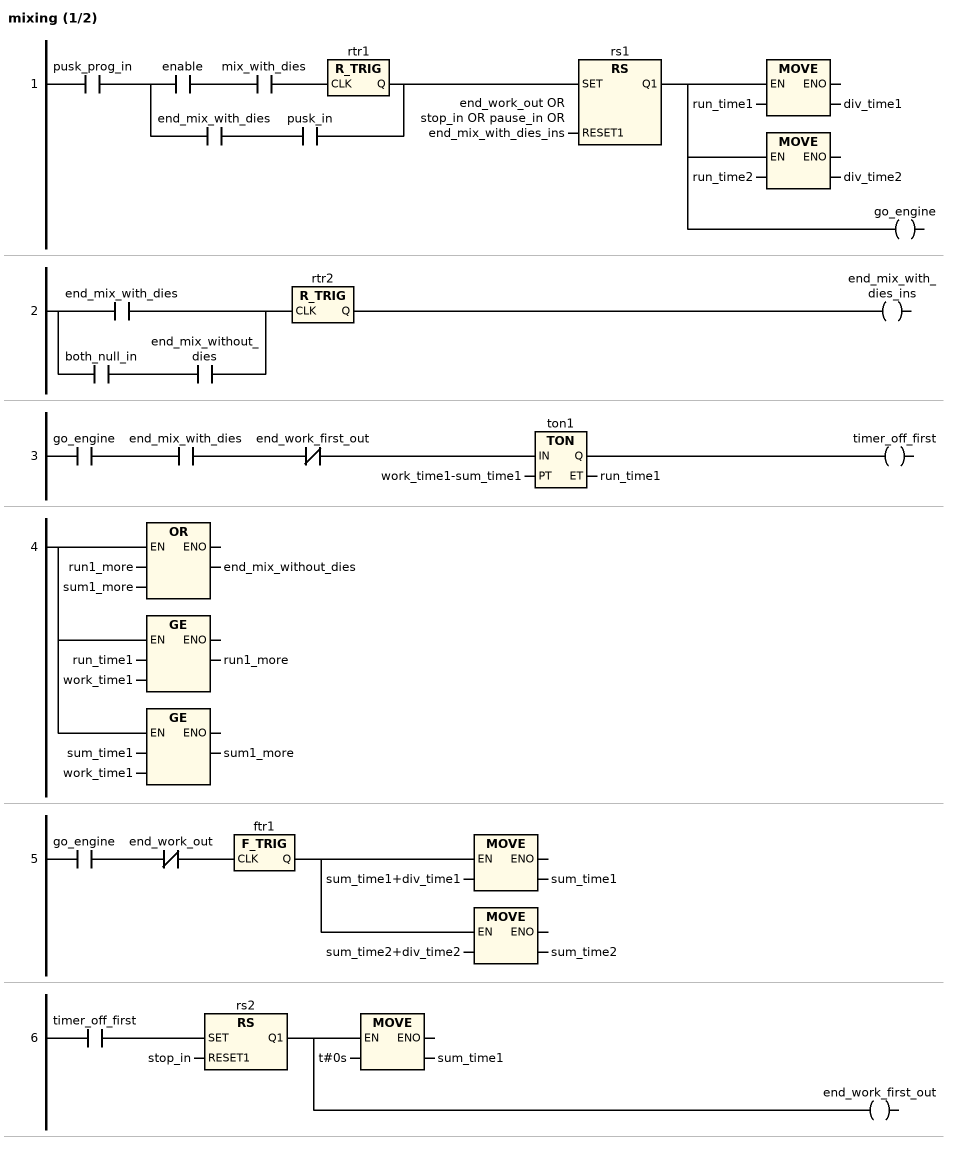
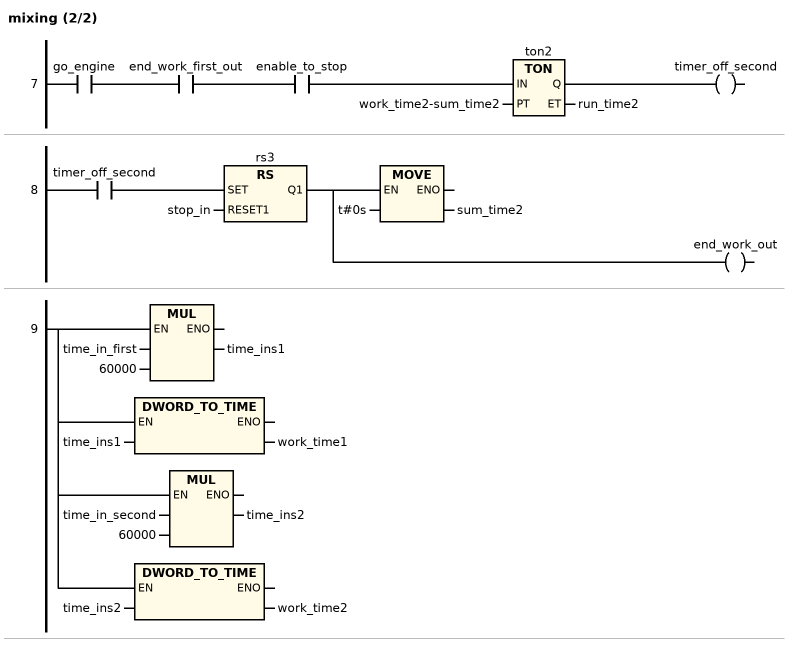
_LD_ (* Ladder Diagram *)
NETWORK 1
	[pusk_prog_in] - { [enable] - [mix_with_dies] - rtr1:R_TRIG(CLK: *) | [end_mix_with_dies] - [pusk_in] } - rs1:RS(SET: *, RESET1: end_work_out OR stop_in OR pause_in OR end_mix_with_dies_ins) --- (go_engine)
		EN --- MOVE(run_time1) => div_time1
		EN --- MOVE(run_time2) => div_time2
NETWORK 2
	{ [end_mix_with_dies] | [both_null_in] - [end_mix_without_dies] } - rtr2:R_TRIG(CLK: *) --- (end_mix_with_dies_ins)
NETWORK 3
	[go_engine] - [end_mix_with_dies] - [/end_work_first_out] - ton1:TON(IN: *, PT: work_time1-sum_time1, ET => run_time1) --- (timer_off_first)
NETWORK 4
	*
		EN --- OR(run1_more, sum1_more) => end_mix_without_dies
		EN --- GE(run_time1, work_time1) => run1_more
		EN --- GE(sum_time1, work_time1) => sum1_more
NETWORK 5
	[go_engine] - [/end_work_out] - ftr1:F_TRIG(CLK: *)
		EN --- MOVE(sum_time1+div_time1) => sum_time1
		EN --- MOVE(sum_time2+div_time2) => sum_time2
NETWORK 6
	[timer_off_first] - rs2:RS(SET: *, RESET1: stop_in) --- (end_work_first_out)
		EN --- MOVE(t#0s) => sum_time1
NETWORK 7
	[go_engine] - [end_work_first_out] - [enable_to_stop] - ton2:TON(IN: *, PT: work_time2-sum_time2, ET => run_time2) --- (timer_off_second)
NETWORK 8
	[timer_off_second] - rs3:RS(SET: *, RESET1: stop_in) --- (end_work_out)
		EN --- MOVE(t#0s) => sum_time2
NETWORK 9
	*
		EN --- MUL(time_in_first, 60000) => time_ins1
		EN --- DWORD_TO_TIME(time_ins1) => work_time1
		EN --- MUL(time_in_second, 60000) => time_ins2
		EN --- DWORD_TO_TIME(time_ins2) => work_time2
_END_LD_
(* the same logic as Structured Text *)
(* Network 1 *)
rtr1(CLK := pusk_prog_in AND enable AND mix_with_dies);
rs1(SET := rtr1.Q OR pusk_prog_in AND end_mix_with_dies AND pusk_in, RESET1 := end_work_out OR stop_in OR pause_in OR end_mix_with_dies_ins);
_p1 := rs1.Q1;
IF _p1 THEN
	div_time1 := run_time1;
	div_time2 := run_time2;
END_IF;
go_engine := _p1;
(* Network 2 *)
rtr2(CLK := end_mix_with_dies OR both_null_in AND end_mix_without_dies);
end_mix_with_dies_ins := rtr2.Q;
(* Network 3 *)
ton1(IN := go_engine AND end_mix_with_dies AND NOT end_work_first_out, PT := work_time1-sum_time1);
run_time1 := ton1.ET;
timer_off_first := ton1.Q;
(* Network 4 *)
end_mix_without_dies := run1_more OR sum1_more;
run1_more := run_time1 >= work_time1;
sum1_more := sum_time1 >= work_time1;
(* Network 5 *)
ftr1(CLK := go_engine AND NOT end_work_out);
IF ftr1.Q THEN
	sum_time1 := sum_time1+div_time1;
	sum_time2 := sum_time2+div_time2;
END_IF;
(* Network 6 *)
rs2(SET := timer_off_first, RESET1 := stop_in);
_p2 := rs2.Q1;
IF _p2 THEN
	sum_time1 := t#0s;
END_IF;
end_work_first_out := _p2;
(* Network 7 *)
ton2(IN := go_engine AND end_work_first_out AND enable_to_stop, PT := work_time2-sum_time2);
run_time2 := ton2.ET;
timer_off_second := ton2.Q;
(* Network 8 *)
rs3(SET := timer_off_second, RESET1 := stop_in);
_p3 := rs3.Q1;
IF _p3 THEN
	sum_time2 := t#0s;
END_IF;
end_work_out := _p3;
(* Network 9 *)
time_ins1 := time_in_first * 60000;
work_time1 := DWORD_TO_TIME(time_ins1);
time_ins2 := time_in_second * 60000;
work_time2 := DWORD_TO_TIME(time_ins2);
END_FUNCTION_BLOCK

(* POU disper, LD *)
FUNCTION_BLOCK disper (*Блок работы насоса диспергатора*)
VAR_INPUT
	pusk_prog_in: BOOL;
	pusk_in: BOOL;
	enable: BOOL;
	stop_in: BOOL;
	pause_in: BOOL;
	weight_in_barrel_in: REAL;
	weight_left: WORD;
END_VAR
VAR_OUTPUT
	go_engine: BOOL;
	end_work: BOOL;
END_VAR
VAR
	rtr1: R_TRIG;
	rs1: RS;
	empty_barrel: BOOL;
	rs2: RS;
	rtr2: R_TRIG;
END_VAR
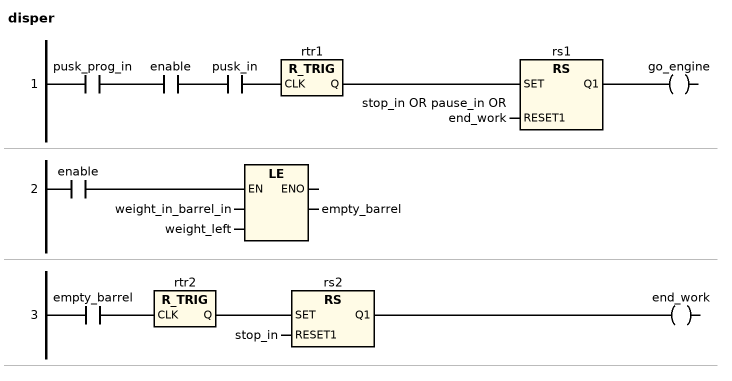
_LD_ (* Ladder Diagram *)
NETWORK 1
	[pusk_prog_in] - [enable] - [pusk_in] - rtr1:R_TRIG(CLK: *) - rs1:RS(SET: *, RESET1: stop_in OR pause_in OR end_work) --- (go_engine)
NETWORK 2
	[enable]
		EN --- LE(weight_in_barrel_in, weight_left) => empty_barrel
NETWORK 3
	[empty_barrel] - rtr2:R_TRIG(CLK: *) - rs2:RS(SET: *, RESET1: stop_in) --- (end_work)
_END_LD_
(* the same logic as Structured Text *)
(* Network 1 *)
rtr1(CLK := pusk_prog_in AND enable AND pusk_in);
rs1(SET := rtr1.Q, RESET1 := stop_in OR pause_in OR end_work);
go_engine := rs1.Q1;
(* Network 2 *)
IF enable THEN
	empty_barrel := weight_in_barrel_in <= weight_left;
END_IF;
(* Network 3 *)
rtr2(CLK := empty_barrel);
rs2(SET := rtr2.Q, RESET1 := stop_in);
end_work := rs2.Q1;
END_FUNCTION_BLOCK
